(*
SPDX-FileCopyrightText: Â© 2026 Oleksandr Tiutyk <trofimich@gmail.com>
SPDX-License-Identifier: MIT
License: https://opensource.org/license/mit
*)

(*!
<summary>Digital output automation component supporting normally-open and normally-closed contacts.</summary>
<description>
Writes evaluated boolean states to physical hardware outputs during the automation output processing phase.
</description>
*)

FUNCTION_BLOCK DigitalOutput EXTENDS TOF_Automation.OutputLeafAutomationComponent
	IMPLEMENTS IDigitalOutput, TOF_Core.IIOBindable
VAR_STAT
	{attribute 'hide'} 
	_ClassName : STRING := __POUNAME();
END_VAR
VAR
	{attribute 'hide'} 
	_ContactType : CONTACT_TYPE;

	_CurrentValue : BOOL;
	_PreviousValue : BOOL;

	_RawValue : REFERENCE TO BOOL;
END_VAR

(*!
<summary>Binds component to a raw boolean process image output variable.</summary>
<param name="rawValue">Reference to physical boolean output variable.</param>
*)
METHOD BindToIO
VAR_INPUT
	rawValue : REFERENCE TO BOOL;
END_VAR
_RawValue REF= rawValue;
END_METHOD

(*!
<summary>Gets whether the component is bound to a valid physical IO variable.</summary>
*)
{attribute 'monitoring' := 'call'}
PROPERTY FINAL BoundToIO : BOOL
GET
BoundToIO := __ISVALIDREF(_RawValue);
END_GET
END_PROPERTY

(*!
<summary>Indicates whether the current logical command differs from the last processed command.</summary>
<description>
ProcessOutput() acknowledges the current command even without an I/O binding.
</description>
*)
{attribute 'monitoring' := 'call'}
PROPERTY FINAL Changed : BOOL
GET
Changed := _CurrentValue <> _PreviousValue;
END_GET
END_PROPERTY

(*!
<summary>Gets the class name of the component.</summary>
*)
{attribute 'monitoring' := 'call'}
PROPERTY ClassName : REFERENCE TO STRING
GET
ClassName REF= _ClassName;
END_GET
END_PROPERTY

(*!
<summary>Gets or sets electrical contact configuration.</summary>
*)
{attribute 'monitoring' := 'call'}
PROPERTY FINAL ContactType : CONTACT_TYPE
GET
ContactType := _ContactType;
END_GET
SET
_ContactType := ContactType;
END_SET
END_PROPERTY

(*!
<summary>Gets the namespace name of the component.</summary>
*)
{attribute 'monitoring' := 'call'}
PROPERTY NamespaceName : REFERENCE TO STRING
GET
NamespaceName REF= CurrentNamespace.Name;
END_GET
END_PROPERTY

(*!
<summary>Writes logical value to the physical output with contact inversion if configured.</summary>
*)
METHOD PROTECTED OnProcessOutput
IF __ISVALIDREF(_RawValue) THEN
	IF _ContactType = CONTACT_TYPE.NORMALLY_CLOSED THEN
		_RawValue := NOT _CurrentValue;
	ELSE
		_RawValue := _CurrentValue;
	END_IF
END_IF

_PreviousValue := _CurrentValue;
END_METHOD

(*!
<summary>Gets the memory size of the instance.</summary>
*)
{attribute 'monitoring' := 'call'}
PROPERTY SelfSize : ULINT
GET
SelfSize := XSIZEOF(THIS^);
END_GET
END_PROPERTY

(*!
<summary>Gets or sets logical boolean state of the output.</summary>
*)
{attribute 'monitoring' := 'call'}
PROPERTY FINAL Value : BOOL
GET
Value := _CurrentValue;
END_GET
SET
_CurrentValue := Value;
END_SET
END_PROPERTY

END_FUNCTION_BLOCK

(* stored: Version 1.1.0.1
   POU DigitalOutput: Id {00c882bb-0de1-4d65-b6f1-d0df694bfb3e}, SpecialFunc None
   Folder Overriden methods: Id {1003a271-38a3-4714-acf5-20b630342852}
   Method BindToIO: Id {b7abc3c5-42d1-477d-92ad-74bb6939db3d}
   Property BoundToIO: Id {9afa4fdb-c488-4031-9bd6-e4df714043e9}
   Get Get: Id {74eac3a2-f493-421c-85c6-0eb55190469f}
   Property Changed: Id {01a5c812-7bcb-40ee-beb8-2111d2bff10d}
   Get Get: Id {7952ae7e-1e32-4e21-ad02-a2b5baf571ff}
   Property ClassName: Id {004ebedb-8d25-4b94-8fe1-e87a1a80e0da}
   Get Get: Id {3febd567-6452-4bd9-9ba7-e16e305a0d7e}
   Property ContactType: Id {52e7a9ab-3a13-457d-99d3-02443f370d77}
   Get Get: Id {5b876d47-6676-47ae-9f28-e36e68801ced}
   Set Set: Id {e996cb3b-a57d-4f8c-8c19-d59088130155}
   Property NamespaceName: Id {336b0713-fd1a-40ad-9ab5-d63a23d7a638}
   Get Get: Id {7fe36426-0451-4643-b7ff-f35ffe55030c}
   Method OnProcessOutput: Id {7b6f0391-82d0-4377-abd0-638493cd0761}
   Property SelfSize: Id {20147cd8-4f58-4ec8-9bf2-efdcff01c0dd}
   Get Get: Id {c04cfb17-d8e5-4f71-829a-687ff94f2753}
   Property Value: Id {848b14c8-ff4e-42f1-84d0-4c9130ca5b8f}
   Get Get: Id {998ae415-763f-4db8-a772-d3ac3df5c5a0}
   Set Set: Id {19530f80-5a6f-4524-910d-5a6d49063051} *)
